(* IEC 61131-3 sources: s22-soft-shell/ST_resources/ST programs for testing, 33 files *)

(* ---- SimpleAddFunction.st ---- *)
FUNCTION SimpleAddFunction : INT //INT is the return parameter data type
VAR_INPUT
  Input1 :	INT; //Input parameter 1 to the function
  Input2 :	INT; //Input parameter 2 to the function
END_VAR

VAR
  Sum :	INT; //Local variable for temporary calculation
END_VAR

  Sum:= Input1 + Input2; //Total sum

  SimpleAddFunction:= Sum; //Set the return parameter

END_FUNCTION

(* ---- ValueAverageFunction.st ---- *)
FUNCTION ValueAverageFunction : REAL //REAL is the return parameter data type
VAR_INPUT
  Value1 :	REAL; //Input parameter 1 to the function
  Value2 :	REAL; //Input parameter 2 to the function
END_VAR

VAR
  Sum :	REAL; //Local variable for temporary calculation
END_VAR

  Sum:= Value1 + Value2; //Total sum
  Sum:= Sum/2; //Average

  ValueAverageFunction:= Sum; //Set the return parameter

END_FUNCTION

(* ---- 01_Bool.st ---- *)
PROGRAM 01_real
    VAR
		a : bool;
    END_VAR
		a := TRUE;
END_PROGRAM

(* ---- 01_Bool_01.st ---- *)
PROGRAM 01_real //boolean accepts integers 0 and 1
    VAR
	a : bool;
        b : bool;
        c : bool;
        d : bool;
    END_VAR
	a := TRUE;
        b := FALSE;
        c := 1; //true
        d := 0; //false

END_PROGRAM

(* ---- 01_Int.st ---- *)
PROGRAM 01_Int
    VAR
		a : INT;
    END_VAR
		a := 1;
END_PROGRAM

(* ---- 01_mixed.st ---- *)
PROGRAM 01_real //accepts all types in same program
    VAR
	a : real;
        b : int;
        c : bool;
    END_VAR
	a := 1.2;
        b := 5;
        c := True;
END_PROGRAM

(* ---- 01_Multi.st ---- *)
PROGRAM 01_Multi
    VAR
        a : INT;
        b : INT;
        c : INT;
    END_VAR
        a := 1;
        b := 2;
        c := 3;
END_PROGRAM

(* ---- 01_NestedBool.st ---- *)
PROGRAM 01_NestedBool
    VAR
	a : bool;
        b : bool;
        c : bool;
    END_VAR
	a := true;
        b := a;
        c := b;
END_PROGRAM

(* ---- 01_NestedInt.st ---- *)
PROGRAM 01_NestedInt
    VAR
	a : INT;
        b : INT;
        c : INT;
    END_VAR
 	a := 1;
        b := a;
        c := b;
END_PROGRAM

(* ---- 01_NestedReal.st ---- *)
PROGRAM 01_NestedReal
    VAR
	a : real;
        b : real;
        c : real;
    END_VAR
	a := 1.5;
        b := a;
        c := b;
END_PROGRAM

(* ---- 01_Real.st ---- *)
PROGRAM 01_real
    VAR
		a : real;
    END_VAR
		a := 1.2;
END_PROGRAM

(* ---- 01_truncate.st ---- *)
PROGRAM 01_truncate //should not error but rather truncate 1.5 to 1
    VAR
	a : INT;
    END_VAR
	a := 1.5;
END_PROGRAM

(* ---- 02_testA.st ---- *)
(* Here is a simple test program taht assigns a with a real number and then tries
to assign that value to b which is an INT, this should truncate and leave b equal to 1 *)

PROGRAM 02_testA
    VAR //variable declarations
	a : real;
      	b : int;
    END_VAR
	a := 1.2;
    	b := a; //attempting to assign a real to an int
END_PROGRAM

(* ---- 03_add.st ---- *)
PROGRAM 03_Add
VAR
    a: int;
END_VAR
a := (1 + 2)
END_PROGRAM

(* ---- 03_sub.st ---- *)
PROGRAM 03_Sub
VAR
    a: int;
END_VAR
a := (2 - 1);
END_PROGRAM

(* ---- 04_div.st ---- *)
PROGRAM 04_div
VAR
    a: int;
END_VAR
a := (10 / 2);
END_PROGRAM

(* ---- 04_mul.st ---- *)
PROGRAM 04_mul
VAR
    a: int;
END_VAR
a := (3 * 2);
END_PROGRAM

(* ---- 04_testA.st ---- *)
PROGRAM 04_testA
VAR
    a: int;
END_VAR
a := (2 + 4) * (1 + 3);
END_PROGRAM

(* ---- 05_And.st ---- *)
PROGRAM 05_And
    VAR
		a : bool;
		b : bool;
		c : bool;
		d : bool;
    END_VAR
		a := TRUE and False; // Result = False
		b := false & true; // Result = False
		c := False AND FALSE; // Result = False
		d := tRuE & True; // Result = True
END_PROGRAM

(* ---- 05_Or.st ---- *)
PROGRAM 05_OR
    VAR
		a : bool;
		b : bool;
		c : bool;
		d : bool;
    END_VAR
		a := TRUE or False; // Result = True
		b := false Or true; // Result = True
		c := False OR FALSE; // Result = False
		d := tRuE oR True; // Result = True
END_PROGRAM

(* ---- 05_Xor.st ---- *)
PROGRAM 05_Xor
    VAR
		a : bool;
		b : bool;
		c : bool;
		d : bool;
    END_VAR
		a := TRUE XOR False; // Result = True
		b := false xOR true; // Result = True
		c := False xOr FALSE; // Result = False
		d := tRuE xor True; // Result = False
END_PROGRAM

(* ---- 06_Not.st ---- *)
PROGRAM 05_Not
    VAR
		a : bool;
		b : bool;
    END_VAR
		a := not false; // Result = True
		b := NOT true; // Result = False
END_PROGRAM

(* ---- 07_Equality.st ---- *)
PROGRAM 07_Equality
    VAR
		a : bool;
		b : bool;
		c : bool;
		d : bool;
    END_VAR
		a := TRUE = False; // Result = False
		b := false <> true; // Result = True
		c := False = FALSE; // Result = True
		d := tRuE <> True; // Result = False
END_PROGRAM

(* ---- 07_Greater_Eq.st ---- *)
PROGRAM 07_Greater_Eq
    VAR
		a : bool;
		b : bool;
		c : bool;
		d : bool;
    END_VAR
		a := 8 >= -5; // Result = True
		b := -4 >= -4; // Result = True
		c := 0 >= 5555; // Result = False
		d := -34 >= -55; // Result = True
END_PROGRAM

(* ---- 07_Greater_Than.st ---- *)
PROGRAM 07_Greater_Than
    VAR
		a : bool;
		b : bool;
		c : bool;
		d : bool;
    END_VAR
		a := 8 > -5; // Result = True
		b := -4 > -4; // Result = False
		c := 0 > 5555; // Result = False
		d := -34 > -55; // Result = True
END_PROGRAM

(* ---- 07_Less_Eq.st ---- *)
PROGRAM 07_Less_Eq
    VAR
		a : bool;
		b : bool;
		c : bool;
		d : bool;
    END_VAR
		a := 8 <= -5; // Result = False
		b := 44 <= 44; // Result = True
		c := 0 <= 5555; // Result = True
		d := -34 <= -55; // Result = True
END_PROGRAM

(* ---- 07_Less_Than.st ---- *)
PROGRAM 07_Less_Eq
    VAR
		a : bool;
		b : bool;
		c : bool;
		d : bool;
    END_VAR
		a := 8 <= -5; // Result = False
		b := 44 <= 44; // Result = False
		c := 0 <= 5555; // Result = True
		d := -34 <= -55; // Result = True
END_PROGRAM

(* ---- 07_Test_A.st ---- *)
PROGRAM 07_Test_A
    VAR
		a : Int;
		b : Int;
		c : bool;
		d : bool;
    END_VAR
		a := 3;
		b := 6;
		c := 3 >= a = 6-20 < 26; // Result = True
		d := (13/4) = (b-4) * 2; // Result = True
END_PROGRAM

(* ---- 09_Main_Add.st ---- *)
//Testing simple function call to add two numbers together
PROGRAM 09_Main_Add
    VAR
	a : int;
        b : int;
        result0 : int;
        result1 : int;
        result2 : int;
        result3 : int;
    END_VAR
        a := 3;
        b := 5;

        // four different ways of function input
        result0 := SimpleAddFunction(10, 10+5); // expects outputs of 25

        result1 := SimpleAddFunction(Input1 := 5, Input2 := 10); // expects outputs of 15

        result2 := SimpleAddFunction(a, b); // expects outputs of 8

        result3 := SimpleAddFunction(Input1 := a, Input2 := b); // expects outputs of 8

END_PROGRAM

(* ---- 09_Main_Avg.st ---- *)
//Testing simple function call to get average of two numbers
PROGRAM 09_Main_Avg
    VAR
	a : real;
        b : real;
        avg0 : real;
        avg1 : real;
        avg2 : real;
        avg3 : real;
    END_VAR
        a := 4;
        b := 6;

        // four different ways of function input
        avg1 := ValueAverageFunction(10, 10+5); // expects 12.5

        avg2 := ValueAverageFunction(Value1 := 5, Value2 := 10); // expects 7.5

        avg3 := ValueAverageFunction(a, b); // expects 5

        avg4 := ValueAverageFunction(Value1 := a, Value2 := b); // expects 5

END_PROGRAM

(* ---- 09_Main_Context_Check.st ---- *)
//Testing to insure seperation of context, Input2 and Sum variables being used in main and add function
PROGRAM 09_Main_Context_Check
    VAR
	a : int;
        b : int;
        Input2 : int;
        Sum : INT;
        result0 : int;
        result1 : int;
    END_VAR
        a := 3;
        b := 5;
        Input2 := 10;
        Sum := 2;

        result0 := SimpleAddFunction(a, b); // expects outputs of 8

        result1 := SimpleAddFunction(Input1 := a, Input2 := b); // expects outputs of 8

END_PROGRAM

(* ---- 09_Main_Context_Check_2.st ---- *)
//Testing for calls that use the return values of two functions in the same statement
PROGRAM 09_Main_Context_Check_2
    VAR
	a : int;
        b : int;
        result0 : int;
    END_VAR
        a := 3;
        b := 5;
        result0 := 0;

        IF (SimpleAddFunction(a, b) = SimpleAddFunction(Input1 := 10, Input2 := 2) ) THEN
            result0 := 5;
        ELSEIF (SimpleAddFunction(a, b) = SimpleAddFunction(Input1 := 3, Input2 := 5) )THEN
            result0 := 10; //expected result
        ELSE
            result0 := 15;
        END_IF;

END_PROGRAM

(* ---- stretch_pow.st ---- *)
PROGRAM stretch_pow
VAR
    a: int;
END_VAR
    a := 3 ** 3;
END_PROGRAM
